{attribute 'OPC.UA.DA' := '0'}
TYPE RFactorBase :
STRUCT
	RFactor_S : LREAL;
	RFactor_P : LREAL;
END_STRUCT
END_TYPE

(* stored: Version 1.1.0.1, ProductVersion 3.1.4024.3
   DUT RFactorBase: Id {36e7baa6-9f7a-417a-ad90-8b4e90f99738} *)
